LIN {X 0,Y 57.012,Z 606.741,A -85,B 0,C 180,E1 -31132.921,E2 -31132.921} C_VEL
LIN {X 0,Y 70.503,Z 602.531,A -85,B 0,C 180,E1 -31135.424,E2 -31135.424} C_VEL
LIN {X 0,Y 77.463,Z 599.719,A -85,B 0,C 180,E1 -31136.349,E2 -31136.349} C_VEL
LIN {X 0,Y 77.371,Z 599.695,A -85,B 0,C 180,E1 -31137.648,E2 -31137.648} C_VEL
LIN {X 0,Y 66.764,Z 603.678,A -85,B 0,C 180,E1 -31139.445,E2 -31139.445} C_VEL
LIN {X 0,Y 56.25,Z 606.589,A -85,B 0,C 180,E1 -31141.785,E2 -31141.785} C_VEL
LIN {X 0,Y 49.306,Z 607.959,A -85,B 0,C 180,E1 -31143.855,E2 -31143.855} C_VEL
LIN {X 0,Y 35.732,Z 609.475,A -85,B 0,C 180,E1 -31150.451,E2 -31150.451} C_VEL
LIN {X 0,Y 24.389,Z 609.412,A -85,B 0,C 180,E1 -31161.943,E2 -31161.943} C_VEL
LIN {X 0,Y 17.702,Z 608.681,A -85,B 0,C 180,E1 -31177.438,E2 -31177.438} C_VEL
LIN {X 0,Y 13.926,Z 607.622,A -85,B 0,C 180,E1 -31199.692,E2 -31199.692} C_VEL
LIN {X 0,Y 14.951,Z 604.796,A -85,B 0,C 180,E1 -31249.904,E2 -31249.904} C_VEL
LIN {X 0,Y 15.875,Z 604.207,A -85,B 0,C 180,E1 -31256.272,E2 -31256.272} C_VEL
LIN {X 0,Y 18.912,Z 602.44,A -85,B 0,C 180,E1 -31271.948,E2 -31271.948} C_VEL
LIN {X 0,Y 24.746,Z 599.09,A -85,B 0,C 180,E1 -31291.276,E2 -31291.276} C_VEL
LIN {X 0,Y 31.926,Z 595.074,A -85,B 0,C 180,E1 -31302.686,E2 -31302.686} C_VEL
LIN {X 0,Y 36.784,Z 592.223,A -85,B 0,C 180,E1 -31305.838,E2 -31305.838} C_VEL
LIN {X 0,Y 46.627,Z 585.645,A -85,B 0,C 180,E1 -31308.441,E2 -31308.441} C_VEL
LIN {X 0,Y 57.037,Z 577.015,A -85,B 0,C 180,E1 -31310.307,E2 -31310.307} C_VEL
LIN {X 0,Y 65.749,Z 568.162,A -85,B 0,C 180,E1 -31311.384,E2 -31311.384} C_VEL
LIN {X 0,Y 73.609,Z 558.428,A -85,B 0,C 180,E1 -31312.119,E2 -31312.119} C_VEL
LIN {X 0,Y 80.58,Z 547.775,A -85,B 0,C 180,E1 -31312.781,E2 -31312.781} C_VEL
LIN {X 0,Y 86.714,Z 535.766,A -85,B 0,C 180,E1 -31313.339,E2 -31313.339} C_VEL
LIN {X 0,Y 91.338,Z 523.82,A -85,B 0,C 180,E1 -31313.786,E2 -31313.786} C_VEL
LIN {X 0,Y 94.81,Z 511.17,A -85,B 0,C 180,E1 -31314.139,E2 -31314.139} C_VEL
LIN {X 0,Y 95.367,Z 508.327,A -85,B 0,C 180,E1 -31314.316,E2 -31314.316} C_VEL
LIN {X 0,Y 95.442,Z 507.971,A -85,B 0,C 180,E1 -31316.07,E2 -31316.07} C_VEL
LIN {X 0,Y 95.333,Z 508.571,A -85,B 0,C 180,E1 -31316.295,E2 -31316.295} C_VEL
LIN {X 0,Y 92.154,Z 521.391,A -85,B 0,C 180,E1 -31316.415,E2 -31316.415} C_VEL
LIN {X 0,Y 88.222,Z 532.433,A -85,B 0,C 180,E1 -31316.666,E2 -31316.666} C_VEL
LIN {X 0,Y 82.697,Z 544.12,A -85,B 0,C 180,E1 -31316.914,E2 -31316.914} C_VEL
LIN {X 0,Y 76.522,Z 554.409,A -85,B 0,C 180,E1 -31317.155,E2 -31317.155} C_VEL
LIN {X 0,Y 68.583,Z 565.071,A -85,B 0,C 180,E1 -31317.569,E2 -31317.569} C_VEL
LIN {X 0,Y 59.76,Z 574.703,A -85,B 0,C 180,E1 -31318.402,E2 -31318.402} C_VEL
LIN {X 0,Y 50.954,Z 582.572,A -85,B 0,C 180,E1 -31319.469,E2 -31319.469} C_VEL
LIN {X 0,Y 42.171,Z 589.094,A -85,B 0,C 180,E1 -31320.799,E2 -31320.799} C_VEL
LIN {X 0,Y 31.705,Z 595.51,A -85,B 0,C 180,E1 -31324.055,E2 -31324.055} C_VEL
LIN {X 0,Y 21.388,Z 600.586,A -85,B 0,C 180,E1 -31329.677,E2 -31329.677} C_VEL
LIN {X 0,Y 11.669,Z 604.517,A -85,B 0,C 180,E1 -31345.395,E2 -31345.395} C_VEL
LIN {X 0,Y 6.082,Z 607.385,A -85,B 0,C 180,E1 -31410,E2 -31410} C_VEL
LIN {X 0,Y 8.949,Z 608.667,A -85,B 0,C 180,E1 -31461.75,E2 -31461.75} C_VEL
LIN {X 0,Y 21.432,Z 610.045,A -85,B 0,C 180,E1 -31489.651,E2 -31489.651} C_VEL
LIN {X 0,Y 28.268,Z 610.141,A -85,B 0,C 180,E1 -31493.962,E2 -31493.962} C_VEL
LIN {X 0,Y 35.211,Z 609.838,A -85,B 0,C 180,E1 -31496.342,E2 -31496.342} C_VEL
LIN {X 0,Y 35.147,Z 609.776,A -85,B 0,C 180,E1 -31498.752,E2 -31498.752} C_VEL
LIN {X 0,Y 28.122,Z 609.97,A -85,B 0,C 180,E1 -31501.591,E2 -31501.591} C_VEL
LIN {X 0,Y 21.198,Z 609.729,A -85,B 0,C 180,E1 -31505.969,E2 -31505.969} C_VEL
LIN {X 0,Y 8.52,Z 608.052,A -85,B 0,C 180,E1 -31534.427,E2 -31534.427} C_VEL
LIN {X 0,Y 9.242,Z 605.026,A -85,B 0,C 180,E1 -31630.477,E2 -31630.477} C_VEL
LIN {X 0,Y 19.296,Z 601.088,A -85,B 0,C 180,E1 -31655.581,E2 -31655.581} C_VEL
LIN {X 0,Y 29.386,Z 596.366,A -85,B 0,C 180,E1 -31663.065,E2 -31663.065} C_VEL
LIN {X 0,Y 36.784,Z 592.223,A -85,B 0,C 180,E1 -31665.838,E2 -31665.838} C_VEL
LIN {X 0,Y 39.722,Z 593.95,A -85,B 0,C 180,E1 -31666.815,E2 -31666.815} C_VEL
LIN {X 0,Y 39.722,Z 600,A -85,B 0,C 180,E1 -31666.815,E2 -31666.815} C_VEL
LIN {X 0,Y 39.722,Z 600,A -85,B 0,C 180,E1 -31666.815,E2 -31666.815}

QRS_NEXT_CUT()

QRS_NEXT()
QRS_HOME()

END
